{attribute 'qualified_only'}
VAR_GLOBAL

	Rotor_RPM_Limit_Exceeded : BOOL; 
	Rotor_RPM_Minimum : REAL;
	Rotor_RPM_Maximum : REAL;
	Rotor_Active_Torque AT %I* : INT;
	

END_VAR

(* stored: Version 1.1.0.1, ProductVersion 3.1.4024.12
   GVL GVL_Rotor: Id {6c2a6d8a-af0d-464f-ab0d-6c6a990188ea} *)
